{attribute addProperty BoxType "EK1100-0000-0018"}
{attribute addProperty Id "Beckhoff_ELM37xxEK1122Beckhoff_ELM37xxEK1122_FB33499C162A_0001_ELM3702_0000_0016ELM3702_1C598C2535244A_0002_ELM3702_0000_0017ELM3702_1C598C2535244A_0003_ELM3704_0000_0016ELM3704_EF18820948060A_0004_ELM3704_0000_0017ELM3704_EF18820948060A_0005_ELM3704_0001_0017ELM3704_EF18820948060A_0006_ELM3704_0020_0016ELM3704_EF18820948060A_0007_ELM3702_0101_0016ELM3702_1C598C2535244A_0008_ELM3704_1001_0016ELM3704_EF18820948060A_0009_ELM3704_1001_0017ELM3704_EF18820948060"}
{attribute addProperty CRC "1490223638"}
{attribute addProperty SizeInBites "3952"}
{attribute addProperty SizeInBytes "494"}
TYPE Beckhoff_ELM37xx_58D30216 EXTENDS EK1100_179A0949 :
STRUCT
	{attribute addProperty Name "Beckhoff_ELM37xxEK1122"}
	Beckhoff_ELM37xxEK1122 : Beckhoff_ELM37xxEK1122_FB33499C;
	{attribute addProperty Name "A_0001_ELM3702_0000_0016"}
	A_0001_ELM3702_0000_0016 : ELM3702_1C598C25;
	{attribute addProperty Name "A_0002_ELM3702_0000_0017"}
	A_0002_ELM3702_0000_0017 : ELM3702_1C598C25;
	{attribute addProperty Name "A_0003_ELM3704_0000_0016"}
	A_0003_ELM3704_0000_0016 : ELM3704_EF188209;
	{attribute addProperty Name "A_0004_ELM3704_0000_0017"}
	A_0004_ELM3704_0000_0017 : ELM3704_EF188209;
	{attribute addProperty Name "A_0005_ELM3704_0001_0017"}
	A_0005_ELM3704_0001_0017 : ELM3704_EF188209;
	{attribute addProperty Name "A_0006_ELM3704_0020_0016"}
	A_0006_ELM3704_0020_0016 : ELM3704_EF188209;
	{attribute addProperty Name "A_0007_ELM3702_0101_0016"}
	A_0007_ELM3702_0101_0016 : ELM3702_1C598C25;
	{attribute addProperty Name "A_0008_ELM3704_1001_0016"}
	A_0008_ELM3704_1001_0016 : ELM3704_EF188209;
	{attribute addProperty Name "A_0009_ELM3704_1001_0017"}
	A_0009_ELM3704_1001_0017 : ELM3704_EF188209;
END_STRUCT
END_TYPE

(* stored: Version 1.2.0.0, ProductVersion 3.1.4024.9
   DUT Beckhoff_ELM37xx_58D30216: Id {9ea24bdd-2b83-4488-b893-d7fbc96129b0} *)
